FUNCTION_BLOCK FB_ReadOnlyStringBuilderAdapter IMPLEMENTS I_ReadOnlyStringBuilderAdapter, I_Enumerable
VAR_INPUT
	ipStringBuilder : I_StringBuilder;
END_VAR

(* Number of bytes allocated in memory for the string builder's contents.*)
PROPERTY Capacity : T_Size
GET
IF THIS^.ipStringBuilder = 0 THEN RETURN; END_IF
Capacity := THIS^.ipStringBuilder.Capacity;
END_GET
END_PROPERTY

(* Copies a subset of characters in the string builder from specified position at specified length to a string*)
METHOD CopySubstringTo : I_ReadOnlyStringBuilderAdapter
VAR_INPUT
	Position, Length : T_Size;
	Value : ANY;
END_VAR
CopySubstringTo := THIS^;
IF THIS^.ipStringBuilder = 0 THEN RETURN; END_IF
THIS^.ipStringBuilder.CopySubstringTo(Position, Length, Value);
END_METHOD

(* Copies contents of string builder to given string of any size*)
METHOD CopyTo : I_ReadOnlyStringBuilderAdapter
VAR_INPUT
	Value : ANY;
END_VAR
CopyTo := THIS^;
IF THIS^.ipStringBuilder = 0 THEN RETURN; END_IF
THIS^.ipStringBuilder.CopyTo(Value);
END_METHOD

(* !!!UNSAFE!!! DON'T FORGET TO RELEASE/DELETE FROM	MEMORY WHEN DONE!
 | Get a copy of the internal string buffer at the size of the string length + 1.*)
METHOD GetBuffer : I_ReadOnlyStringBuilderAdapter
VAR_IN_OUT
	pBuffer	: POINTER TO BYTE;
END_VAR
GetBuffer := THIS^;
IF THIS^.ipStringBuilder = 0 THEN RETURN; END_IF
THIS^.ipStringBuilder.GetBuffer(pBuffer);
END_METHOD

(* Retrieves the number of bytes allocated in memory for the string builder's contents.*)
METHOD GetCapacity : I_ReadOnlyStringBuilderAdapter
VAR_OUTPUT
	Capacity	: T_Size;
END_VAR
GetCapacity := THIS^;
Capacity := THIS^.Capacity;
END_METHOD

(* Gets character at specified position in the string builder*)
METHOD GetChar : T_Char
VAR_INPUT
	Position	: T_Size;
END_VAR
IF THIS^.ipStringBuilder = 0 THEN RETURN; END_IF
GetChar := THIS^.ipStringBuilder.GetChar(Position);
END_METHOD

METHOD GetEnumerator : I_Enumerator
VAR_INST
	fbEnumerator : FB_StringBuilderEnumerator(THIS^.ipStringBuilder);
END_VAR
fbEnumerator.FB_init(0,0,THIS^.ipStringBuilder);
GetEnumerator := fbEnumerator;
END_METHOD

(* Retrieves the current size of string builder contents*)
METHOD GetLength : I_ReadOnlyStringBuilderAdapter
VAR_OUTPUT
	Length	: T_Size;
END_VAR
GetLength := THIS^;
Length := THIS^.Length;
END_METHOD

(* Converts contents of string builder to string and returns them*)
METHOD GetString : T_LongString
IF THIS^.ipStringBuilder = 0 THEN RETURN; END_IF
GetString := THIS^.ipStringBuilder.GetString();
END_METHOD

(* Get a subset of characters in the string builder from specified position at specified length and returns them as a string*)
METHOD GetSubstring : T_LongString
VAR_INPUT
	Position	: T_Size;
	Length	: T_Size;
END_VAR
IF THIS^.ipStringBuilder = 0 THEN RETURN; END_IF
GetSubstring := THIS^.ipStringBuilder.GetSubstring(Position, Length);
END_METHOD

(* Current size of string builder contents*)
PROPERTY Length : T_Size
GET
IF THIS^.ipStringBuilder = 0 THEN RETURN; END_IF
Length := THIS^.ipStringBuilder.Length;
END_GET
END_PROPERTY

(* Finds the position of the first instance of a given string in the content's of the string builder from a starting position*)
METHOD Search : I_ReadOnlyStringBuilderAdapter
VAR_INPUT
	sValue	: T_LongString;
	Start_Position	: T_Size;
END_VAR
VAR_OUTPUT
	Position	: T_Size;
END_VAR
Search := THIS^;
IF THIS^.ipStringBuilder = 0 THEN RETURN; END_IF
THIS^.ipStringBuilder.Search(sValue, Start_Position, Position => Position);
END_METHOD

(* Finds the position of the first instance of a given value in the content's of the string builder from a starting position*)
METHOD SearchAny : I_ReadOnlyStringBuilderAdapter
VAR_INPUT
	Value : ANY;
	Start_Position : T_Size;
END_VAR
VAR_OUTPUT
	Position : T_Size := -1;
END_VAR
SearchAny := THIS^;
IF THIS^.ipStringBuilder = 0 THEN RETURN; END_IF
THIS^.ipStringBuilder.SearchAny(Value, Start_Position, Position => Position);
END_METHOD

(* Appends selected characters from the current string builder to the selected string builder*)
METHOD Split : I_ReadOnlyStringBuilderAdapter
VAR_INPUT
	Position, Length : T_Size;
	ipStringBuilder : I_StringBuilder;
END_VAR
Split := THIS^;
IF THIS^.ipStringBuilder = 0 THEN RETURN; END_IF
THIS^.ipStringBuilder.Split(Position, Length, ipStringBuilder);
END_METHOD

END_FUNCTION_BLOCK

(* stored: Version 1.1.0.1, ProductVersion 3.1.4024.4
   POU FB_ReadOnlyStringBuilderAdapter: Id {5b2f76d6-71b2-41fd-9735-b5916830d938}, SpecialFunc None
   Property Capacity: Id {5e804c55-c620-4d22-a532-fbaedf7e33f3}
   Get Get: Id {a02353a6-8f43-4024-b756-1b601822b353}
   Method CopySubstringTo: Id {e52e47a2-b7cb-4fc2-937d-d79a7dd6f1c1}
   Method CopyTo: Id {cd0ca31a-3a35-4a56-9e9a-84c2c0a452e5}
   Method GetBuffer: Id {0e58de1f-9791-406a-84d4-e5bae5496810}
   Method GetCapacity: Id {e0b2a79e-d112-46c1-a77e-9c5f7b9fc05b}
   Method GetChar: Id {1af0a8ac-26b2-40b7-8c19-3ef6ce240260}
   Method GetEnumerator: Id {55b67b81-ce26-456d-b5b2-4ac663be4f03}
   Method GetLength: Id {84f2c33b-4773-4941-aceb-9877e5a12da1}
   Method GetString: Id {65690ebe-27e3-45fa-ab0e-48130b75ef40}
   Method GetSubstring: Id {9fa3ecbe-5e9c-4351-b490-0efbc9d44201}
   Property Length: Id {47428ebe-0553-4546-9fa2-3c3da99dd0e5}
   Get Get: Id {f03399eb-acc0-45e6-b564-02633cd162e1}
   Method Search: Id {cad7533e-4311-4c28-a285-5b01561ebfe0}
   Method SearchAny: Id {67b278b9-ea26-4100-9ab4-f6713e4518df}
   Method Split: Id {90821461-a891-4b50-8400-5b7b505302ad} *)
